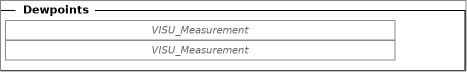
VISUALIZATION VISU_TelemetryDewpoints  // 467x72
VAR_IN_OUT
    ref : TelemetryDewpoints;
	widget : TelemetryDewpointsWidget;
END_VAR
    Label (20,0 75x20), "Dewpoints"
    Line (465,70) (465,10)
        p2175578022: widget.actualStatus.color.bg
    Frame (5,20 390x20)
        shows VISU_Measurement(widget := widget.topAir)
    Frame (5,40 390x20)
        shows VISU_Measurement(widget := widget.insideTube)
    Line (95,10) (465,10)
        p2175578022: widget.actualStatus.color.bg
    Line (0,10) (15,10)
        p2175578022: widget.actualStatus.color.bg
    Line (0,70) (0,10)
        p2175578022: widget.actualStatus.color.bg
    Line (0,70) (465,70)
        p2175578022: widget.actualStatus.color.bg
END_VISUALIZATION

(* stored: Version 1.1.0.1, ProductVersion 3.1.4019.2
   Visu VISU_TelemetryDewpoints: Id {c5d84449-5948-436c-bf83-cb9b68b6b3e8} *)
